FUNCTION ValidateInterface : Result
VAR_INPUT
	iToValidate: I_ValidateInterface;
END_VAR
VAR
	_err: __SYSTEM.ExceptionCode;
END_VAR

IF iToValidate = 0 THEN
	ValidateInterface := Error;
	RETURN;
END_IF

__TRY
	iToValidate.ValidateInterface();
	ValidateInterface := Ok;
__CATCH(_err)
	ValidateInterface := Error;
__ENDTRY

END_FUNCTION

(* stored: Version 1.1.0.1
   POU ValidateInterface: Id {0e731eaf-cbba-483d-8555-81138479f57f}, SpecialFunc None *)
